Staubli VAL3: setFrameId.pgx

public program setFrameId(num x_nIndex)
  local num i
begin
  //
  // save the FrameId
  //
  pEditPoint.nIndexFrame=x_nIndex
  // link to the father frame and alll the point
  link(pEditPoint.fFrame,saveData:fFrameItem[x_nIndex].fFrame)
  for i=0 to size(pEditPoint.tData)-1
    link(pEditPoint.tData[i].pPoint,pEditPoint.fFrame)
  endFor
end
